// TIA Portal V16 export
// export: Created 2024-09-05T17:39:17.4635556Z, ExportSetting WithDefaults, DisplayName Totally Integrated Automation Portal, DisplayVersion V16 Update 6, DisplayName TIA Portal Version Control Interface, DisplayVersion V16 Update 2, DisplayName TIA Portal Openness, DisplayVersion V16 Update 6, DisplayName STEP 7 Professional, DisplayVersion V16 Update 6, DisplayName STEP 7 Safety, DisplayVersion V16, DisplayName WinCC Advanced, DisplayVersion V16 Update 6
DATA_BLOCK "ProductionProgramCounters_DB"   // DB67
VERSION : 0.1
// stored: AutoNumber true, DBAccessibleFromOPCUA true, InstanceOfName ProductionProgramCounters, InstanceOfType FB
"ProductionProgramCounters"
   // VAR
   //    referenceOld : Int := 1;
   //    shiftToDelete : Int := 0;
   // END_VAR
BEGIN
END_DATA_BLOCK
